(* CODESYS project BelShina_8100_1_1_1.export

Project tree, tasks and I/O mapping:
  application Application
    libraries: ; WagoAppStepper, 1.6.1.1 (WAGO)
    task PLC_Task (cyclic, interval t#50ms, priority 15) calls PLC_PRG
    DataTypes/
      data type ConturBuffer
      data type CurveStates
      data type ForceStepStates
      data type StepperStates
      data type StiffnessTestStates
    GV/
      global variables AI_Sensors
      global variables HMI_Alm
      global variables HMI_Process
      global variables HMI_Stepper
    Program/
      Device/
        Motors/
          ForceStep/
            function block fbForceStep [ST]: METH_Direction
            function block fbGetKoef [ST]
            function block fbSpeedCalc [ST]
            program prForceStep [ST]
          Stepper/
            function block fbStepper [ST]: ACT_MoveHome, ACT_MoveToPos, METH_Direction
            program prLaserStepper_1 [ST]
            program prLaserStepper_2 [ST]
          program prMotion [ST]
        program prDevice [ST]
      IO/
        function block filter [ST]
        function fnoneDigit [ST]
        function fnUpToTen [ST]
        function fnZeroDigit [ST]
        program prInToVars [ST]
      OPC_Sync/
        function block fbReadBuffOPC [ST]
        function block FillBuffer [ST]
      Process/
        GetCurve/
          function block fbGetCurve [ST]
          program prGetCurve_1 [ST]
          program prGetCurve_2 [ST]
          program prGetCurve_2_2 [ST]
        StiffnessTest/
          function block fbCalcDistance [ST]
          function block fbStiffnessTest [ST]
          program prStiffnessTest_1 [ST]
          program prStiffnessTest_2 [ST]
        program prProcess [ST]
      function block LIN_TRAFO [ST]
    Simulation/
      function block fbForceStepSim [ST]
      function block fbStepperSim [ST]
      program prSimulation [ST]
    program PLC_PRG [ST]
    Symbols
*)

// Application/DataTypes/ConturBuffer
TYPE ConturBuffer :
STRUCT
	arStepPos			: ARRAY[0..600] OF REAL;
	arLaserData			: ARRAY[0..600] OF REAL;
	wIndex			: WORD;
	xDone			: BOOL;
	 
END_STRUCT
END_TYPE

// Application/DataTypes/CurveStates

TYPE CurveStates :
(
	CS_Stop 		:= 0,
	CS_Done			:= 1,
	CS_Stopping		:= 2,
	CS_SetStep		:= 3,
	CS_WaitInitial	:= 4,
	CS_SetMeassure	:= 5,
	CS_Measuring	:= 6,
	CS_ReadingOPC	:= 7
);
END_TYPE

// Application/DataTypes/ForceStepStates

TYPE ForceStepStates :
(
	FS_Stop 				:= 0,
	FS_FirstRun 			:= 1,
	FS_WaitRaughApprox		:= 2,
	FS_MakeStep				:= 3,
	FS_CheckForce			:= 4,
	FS_Done					:= 5,
	FS_StartRelease			:= 6,
	FS_WaitRelease			:= 7,
	FS_MovePos				:= 8,
	FS_WaitVelicity			:= 9,
	FS_VelicityMode			:= 10,
	FS_VelicityStopping		:= 11
);
END_TYPE

// Application/DataTypes/StepperStates

TYPE StepperStates :
(
	SM_Idle 			:=0,
	SM_Homing			:=1,
	SM_HommingRough		:=2,
	SM_Home				:=3,
	SM_SetZeroPos		:=4,
	SM_SetPrm			:=5,
	SM_MovingToPos		:=6,
	SM_OnPos			:=7,
	SM_Stopping 		:=8,
	SM_Stop 			:=9
);
END_TYPE

// Application/DataTypes/StiffnessTestStates

TYPE StiffnessTestStates :
(
	ST_Proc_Stop 			:= 0,
	ST_Proc_GettingForce 	:= 1,
	ST_Proc_GettingHalfKoef	:= 2,
	ST_Proc_CalcKoef		:= 3,
	ST_Proc_GettingCurve	:= 4,
	ST_Proc_Done			:= 5,
	ST_Proc_Releasing		:= 6,
	ST_Proc_Stopping		:= 7,
	ST_Proc_GettingFirstCurve:=8,
	ST_Proc_Pause			:= 9,
	ST_SendingData			:=10
	
);
END_TYPE

// Application/GV/AI_Sensors

VAR_GLOBAL
	AI_Rol_1 		AT %IW1 : WORD;
	AI_Rol_2 		AT %IW2 : WORD;
	AI_Laser_1 		AT %IW3 : WORD;
	AI_Laser_2 		AT %IW4 : WORD;
	
	wCounter_1		AT %IW29 : WORD;
	wCounter_2		AT %IW31 : WORD;
	dwCounter		: DWORD;
	Force_Us		AT %IW32 : WORD;
	Force_Ref		AT %IW33 : WORD;
	
	FS_Status_1_1		AT %IB41 : BYTE;
	FS_Status_1_2		AT %IB42 : BYTE;
	FS_Status_1_3		AT %IB43 : BYTE;
	
	FS_Status_Force_3		AT %IB29 : BYTE;
	FS_Status_Force_3_2		AT %IB31 : BYTE;
	
	FS_Status_2_1		AT %IB53 : BYTE;
	FS_Status_2_2		AT %IB54 : BYTE;
	FS_Status_2_3		AT %IB55 : BYTE;
	
	Contr_0		AT %QB38 : BYTE;
	Contr_1		AT %QB42 : BYTE;
	SetPos		AT %QW20 : WORD;
	
	
	
	xStopSwitchLeft: BOOL;
	xStopSwitchRight: BOOL;
	
	LaserHome_1: BOOL;
	LaserHome_2: BOOL;
	LaserUp_1: 	BOOL;
	LaserUp_2:	BOOL;
	
	
	xGlWrite1		:BOOL;
	xGlWrite2		:BOOL;
	
END_VAR

// Application/GV/HMI_Alm

VAR_GLOBAL
	xResetAlm		: BOOL;
	wForceStepAlm	: WORD;
	wAnyAlm			: WORD;
	wAlmLaser_1		: WORD;
	wAlmLaser_2		: WORD;
END_VAR

// Application/GV/HMI_Process

VAR_GLOBAL
	///////////////////////////   GET CURVE 1  //////////////////////
	
	xGC_Start_1: BOOL;
	wGS_State_1: WORD;
	
	///////////////////////////   GET CURVE 2  //////////////////////
	
	xGC_Start_2: BOOL;
	wGS_State_2: WORD;
	
	////////////////////////////  STIFFNESS TEST 1 /////////////////////////////
	
	xGS_StartProc_1: BOOL;
	wST_State_1: WORD;
	rST_Koef_1: REAL;
	wST_HalfPos_1: REAL;
	wST_HalfForce_1: REAL;
	xST_Ready_1: BOOL;
	rST_Way_1:REAL;
	rST_Force_1: REAL;
	xStartAllCurves:	BOOL;
	
	////////////////////////////  STIFFNESS TEST 2 /////////////////////////////
	
	xGS_StartProc_2: BOOL;
	wST_State_2: StiffnessTestStates;
	rST_Koef_2: REAL;
	wST_HalfPos_2: REAL;
	wST_HalfForce_2: REAL;
	xST_Ready_2: BOOL;
	rST_Way_2:REAL;
	rST_Force_2: REAL;
	
	////////////////////////////  STIFFNESS TEST 3 /////////////////////////////
	
	xGS_StartProc_3: BOOL;
	wST_State_3: StiffnessTestStates;
	rST_Koef_3: REAL;
	wST_HalfPos_3: REAL;
	wST_HalfForce_3: REAL;
	xST_Ready_3: BOOL;
	rST_Way_3:REAL;
	rST_Force_3: REAL;
	
	////////////////////////////  DISTANCE /////////////////////////////
	
	rDistance_1		: REAL;
	rDistance_2		: REAL;
	
	rTablePos_1		: REAL;
	rTablePos_2		: REAL;
	rLaserDistance_1		: REAL;
	rLaserDistance_2		: REAL;
	
	xProcFinished			: BOOL;
	wProcType	: WORD;
	xReadOPC_1:	BOOL;
	xReadOPC_2:	BOOL;
	xCurveStarted_1: BOOL;
	xCurveStarted_2: BOOL;
	
	rStepPos_1:	REAL;
	rStepPos_2:	REAL;
	
	rLaserData_1: REAL;
	rLaserData_2: REAL;
	
	wBufferState_1:	WORD;
	wBufferState_2:	WORD;
	
	xContinue:	BOOL;
	
	rRealGetForce:	REAL;
	rRealGetForceMax:	REAL;
	diDistanceForce:	DINT;
	
END_VAR
VAR_GLOBAL RETAIN
	///////////////////////////   GET CURVE 1  //////////////////////
	
	wGC_Distance_1: WORD;
	wGC_InitialPos_1: WORD;
	wGC_EndPos_1: WORD;
	
	///////////////////////////   GET CURVE 2  //////////////////////
	
	wGC_Distance_2: WORD;
	wGC_InitialPos_2: WORD;
	wGC_EndPos_2: WORD;
	
	////////////////////////////  STIFFNESS TEST 1 /////////////////////////////
	
	rST_GetForce_1: REAL;
	rST_SetForce_1: REAL;
	wGS_WaitTillDone_1: WORD;
	
	////////////////////////////  STIFFNESS TEST 2 /////////////////////////////
	
	rST_GetForce_2: REAL;
	rST_SetForce_2: REAL;
	wGS_WaitTillDone_2: WORD;
	
	rKforce_1:	REAL:=1; // попроавка на элластичность троса
	rKforce_2:	REAL:=1; // попроавка на элластичность троса
	rKforce_Ctcle:	REAL:=1; // попроавка на элластичность троса
	rRadius:	REAL:=1;
	
	
	
	wTyreSizeFirst:	WORD;
	wTyreSizeAfter:	WORD;
	
	rCycleForceOffset:	REAL;
	rLineForceOffset_1:	REAL;
	rLineForceOffset_2:	REAL;
	
	rDistanceBetweenLasers:	REAL:=1300;
	
	rLaserSetPos_1:	REAL;
	rLaserSetpos_2:	REAL;
	
END_VAR

// Application/GV/HMI_Stepper

VAR_GLOBAL
	///////////////////////    FORCE STEP    //////////////////////////////
	rFS_GetForce: REAL;	
	xFS_Start: BOOL;
	xFS_Release: BOOL;
	wFS_State: WORD;
	wFS_ActualPos: DWORD;
	xFS_JogLeft: BOOL;
	xFS_JogRight: BOOL;
	rFS_GetForce_check: REAL;	
	rFS_CycledWay:	REAL;
	rFS_LinedWay_1:	REAL;
	rFS_LinedWay_2:	REAL;
	rAngle: REAL;
	
	
	///////////////////////////   LASER  STEP 1  //////////////////////
	xLS_MoveToPos_1: BOOL;
	xLS_MoveHome_1: BOOL;
	xLS_Stop_1: BOOL;
	wLS_GetPos_1: DINT;
	wLS_StepperState_1: WORD;
	xLS_Initilized_1: BOOL;
	rLS_RealPos_1:	REAL;
	
	///////////////////////////   LASER  STEP 2  //////////////////////
	xLS_MoveToPos_2: BOOL;
	xLS_MoveHome_2: BOOL;
	xLS_Stop_2: BOOL;
	wLS_GetPos_2: DINT;
	wLS_StepperState_2: WORD;
	xLS_Initilized_2: BOOL;
	rLS_RealPos_2:	REAL;
	
	
	
END_VAR
VAR_GLOBAL RETAIN
	
///////////////////////    FORCE STEP    //////////////////////////////
	rFS_SetForce: REAL;
	wFS_RoughApprox: WORD;
	wFS_Step: WORD;
	xFS_DirNeg: BOOL;
	rFS_Sensativity: REAL;
	wFS_SetSpeed: WORD;
	wFS_SetAcceleration: WORD;
	wFS_SetDeceleration: WORD;
	wFS_SetBackSpeed: WORD;
	
	
///////////////////////////   LASER  STEP 1  //////////////////////	
	wLS_SetPos_1: WORD;
	wLS_SetSpeed_1: WORD;
	xLS_DirNeg_1: BOOL;
	wLS_Acceleration_1: WORD;
	wLS_Deceleration_1: WORD;
	xLS_StandStill_1:	BOOL;
	
	///////////////////////////   LASER  STEP 2  //////////////////////	
	wLS_SetPos_2: WORD;
	wLS_SetSpeed_2: WORD;
	xLS_DirNeg_2: BOOL;
	wLS_Acceleration_2: WORD;
	wLS_Deceleration_2: WORD;
	xLS_StandStill_2:	BOOL;
	
	
	k_1: REAL:=0.00763;
	k_2: REAL:=0.00763;
	k_3: REAL:=0.0198;
	k_4: REAL:=0.0198;
	
	StepAngle_1:	REAL:=1.8;
	StepAngle_2:	REAL:=1.8;
	ScrewStep_1:	REAL:=24;
	ScrewStep_2:	REAL:=24;
	
	ScrewStepForce:	REAL:=5;
	
	rReductCoef:	REAL:=1;
	rStepAngleForce:	REAL:=1.8;
	
	rForceSensorScale:	REAL:= 20000;
	
	rEncoderImpulseCount: WORD:=5000;
	
	
	
	
	
	
	
	
	
END_VAR

// Application/PLC_PRG
PROGRAM PLC_PRG
VAR
	tnAlmReset:	TON;
	tnStop_1:	TON;
	tnStop_2:	TON;
END_VAR

prInToVars();
prDevice();
prProcess();
tnAlmReset(IN:=xResetAlm, PT:= T#3S);
IF tnAlmReset.Q THEN
	xResetAlm:= FALSE;
END_IF
tnStop_1(IN:=xLS_Stop_1, PT:= T#3S);
IF tnAlmReset.Q THEN
	xLS_Stop_1:= FALSE;
END_IF
tnStop_2(IN:=xLS_Stop_1, PT:= T#3S);
IF tnAlmReset.Q THEN
	xLS_Stop_2:= FALSE;
END_IF
//xResetAlm:=FALSE;
//prSimulation();
//xLS_Stop_1

END_PROGRAM

// Application/Program/IO/prInToVars
PROGRAM prInToVars
	
VAR
	
	_LaserDistance_1: REAL;
	_LaserDistance_2: REAL;
	TRAFO:LIN_TRAFO;
	TRAFO_1:LIN_TRAFO;
	Ud : REAL;
	Uv:	REAL;
	
	filter_1: filter;
	filter_2: filter;
	filter_force: filter;
	k1:	REAL:=0.97;
	k2: REAL:=0.9;
	k_force:REAL:=0.9;
	xSetZero: BOOL;
	rtForceStart:	R_TRIG;
	rtScanStart:	R_TRIG;
	ftContinue:	F_TRIG;
	rtRead1:	F_TRIG;
	rtRead2:	F_TRIG;
	xRef:	BOOL;
	rForceLoc:	REAL;
	rtGetInitialPos:	R_TRIG;
	rOldDistance:	real;
END_VAR

//rDistance_1 := TO_REAL(AI_Rol_1) * k_1;
//rDistance_2 := TO_REAL(AI_Rol_2) * k_2;

rTablePos_1:= TO_REAL(AI_Rol_1) * k_1;
rTablePos_2:= TO_REAL(AI_Rol_2) * k_2;
rTablePos_1:=fnoneDigit(in:= rTablePos_1);
rTablePos_2:=fnoneDigit(in:= rTablePos_2);
//rLaserDistance_1 := 150 + TO_REAL(AI_Laser_1) * k_3;

//rLaserDistance_2 := 150 + rDistanceBetweenLasers - TO_REAL(AI_Laser_2) * k_3;
rtGetInitialPos(CLK:= wGS_State_1 > CS_WaitInitial AND wGS_State_2 > CS_WaitInitial,);
(*IF rtGetInitialPos.Q THEN
	rDistanceBetweenLasers:= (150 + TO_REAL(AI_Laser_1) * k_3) + (150 + TO_REAL(AI_Laser_2) * k_3) + (rRadius * 2);
END_IF*)
_LaserDistance_1:= 150 + TO_REAL(AI_Laser_1) * k_3;
_LaserDistance_2:= rDistanceBetweenLasers - (TO_REAL(AI_Laser_2) * k_3 + 150) - rLaserSetPos_1 - rLaserSetPos_2;
rtScanStart(CLK:= xStartAllCurves); // xContinue
ftContinue(CLK:=xContinue);
rtRead1(CLK:=wLS_StepperState_1 = SM_OnPos);
rtRead2(CLK:=wLS_StepperState_2 = SM_OnPos);
(*
IF wGS_State_1 = CS_WaitInitial OR  rtRead1.Q OR wST_State_1 = ST_Proc_Done OR wST_State_1 = SM_Stop THEN
	//xGlWrite1:=FALSE;
	//filter_1(F_IN:= rDistance_1);
	filter_1(F_IN:= _LaserDistance_1, k:= k1, F_OUT=> rLaserDistance_1);
END_IF
IF wGS_State_2 = CS_WaitInitial OR rtRead2.Q OR wST_State_1 = ST_Proc_Done OR wST_State_1 = SM_Stop THEN
	//xGlWrite2:=FALSE;
	//filter_2(F_IN:= rDistance_2);
	filter_2(F_IN:= _LaserDistance_2, k:= k1,F_OUT=> rLaserDistance_2);
END_IF
*)
filter_1(F_IN:= _LaserDistance_1, k:= k1, F_OUT=> rLaserDistance_1);
filter_2(F_IN:= _LaserDistance_2, k:= k1,F_OUT=> rLaserDistance_2);
rLaserDistance_1:=fnoneDigit(rLaserDistance_1);
rLaserDistance_2:=fnoneDigit(rLaserDistance_2);

//filter_1(F_IN:= rDistance_1, k:= k1, F_OUT=> rLaserDistance_1);
//filter_2(F_IN:= rDistance_2, k:= k1,F_OUT=> rLaserDistance_2);

TRAFO(
	IN:= TO_REAL(Force_Us), 
	IN_MIN:= 0, 
	IN_MAX:= 30000, 
	OUT_MIN:= 0, 
	OUT_MAX:= 15, 
	OUT=> , 
	ERROR=> );
	filter_force(F_IN:= TRAFO.OUT, k:= k_force, F_OUT=> Ud);
	TRAFO_1(
	IN:= TO_REAL(Force_Ref), 
	IN_MIN:= 0, 
	IN_MAX:= 20000, 
	OUT_MIN:= 0, 
	OUT_MAX:= 10, 
	OUT=> Uv, 
	ERROR=> );

	
CASE wProcType OF
	1:
		rFS_GetForce:= (((Ud/2)/(Uv))*rForceSensorScale + rCycleForceOffset) * rKforce_Ctcle * rRadius;
		rFS_GetForce:=fnUpToTen(rFS_GetForce);
		IF (rFS_CycledWay <> rOldDistance) THEN
			rOldDistance:= rFS_CycledWay;
			diDistanceForce:= TO_DINT(rFS_GetForce) * 10000 + TO_DINT(rFS_CycledWay*100);
		END_IF
		
	2:
		rFS_GetForce:= (((Ud/2)/(Uv))*rForceSensorScale + rLineForceOffset_1)* rKforce_1;
		rFS_GetForce:=fnUpToTen(rFS_GetForce);
		IF (rDistance_1 <> rOldDistance) THEN
			rOldDistance:= rDistance_1;
			diDistanceForce:= TO_DINT(rFS_GetForce) * 10000 + TO_DINT(rDistance_1 *100);
		END_IF
		
	3:
		rFS_GetForce:= (((Ud/2)/(Uv))*rForceSensorScale + rLineForceOffset_2) * rKforce_2;
		rFS_GetForce:=fnUpToTen(rFS_GetForce);
		IF (rDistance_2 <> rOldDistance) THEN
			rOldDistance:= rDistance_2;
			diDistanceForce:= TO_DINT(rFS_GetForce) * 10000 + TO_DINT(rDistance_2 *100);
		END_IF
		
END_CASE
//rFS_GetForce:=fnZeroDigit(in:= rFS_GetForce);
//rRealGetForce:= ((Ud/2)/(Uv))*rForceSensorScale * rKforce_1;
//rRealGetForce:=fnZeroDigit(rRealGetForce);
rRealGetForce:= rFS_GetForce / rRadius;
rRealGetForce:= fnUpToTen(rRealGetForce);
rRealGetForceMax:= rST_Force_1 / rRadius;
rRealGetForceMax:= rRealGetForce;

xLS_StandStill_1:=AI_Sensors.FS_Status_1_2.2;
xLS_StandStill_2:=AI_Sensors.FS_Status_2_2.2;

dwCounter:= wCounter_2 * 68835 + wCounter_1;
rAngle:= ((TO_REAL(dwCounter)) / (TO_REAL(rEncoderImpulseCount)) * 90);
rAngle:=fnoneDigit(rAngle);

//xFS_Start
rtForceStart(CLK:=xGS_StartProc_1);

IF rtForceStart.Q THEN
	SetPos:= 5000;
	Contr_0.2:=TRUE;
ELSE
	Contr_0.2:=FALSE;
END_IF

xRef:= FS_Status_Force_3.1;

(*
xStopSwitchLeft:= NOT FS_Status_Force_3.1;
xStopSwitchRight:= NOT FS_Status_Force_3_2.1;

LaserHome_1:= NOT FS_Status_Force_3.1;
LaserHome_2:= NOT FS_Status_Force_3_2.1;

LaserUp_1:= NOT FS_Status_Force_3.4;
LaserUp_2:= NOT FS_Status_Force_3_2.4;
*)

//xSetZero:=FALSE;

END_PROGRAM

// Application/Program/IO/fnoneDigit
FUNCTION fnoneDigit : REAL
VAR_INPUT
	in: REAL;
END_VAR
VAR
	iBuffer:	INT;
	out:	REAL;
END_VAR

iBuffer:= TO_INT(in * 10);
out:=TO_REAL(iBuffer)/10;
fnoneDigit:=out;

END_FUNCTION

// Application/Program/IO/fnUpToTen
FUNCTION fnUpToTen : REAL
VAR_INPUT
	in: REAL;
END_VAR
VAR
	iBuffer:	INT;
	out:	REAL;
END_VAR

iBuffer:= TO_INT(in/10);
out:=iBuffer*10;
fnUpToTen:=out;

END_FUNCTION

// Application/Program/IO/fnZeroDigit
FUNCTION fnZeroDigit : REAL
VAR_INPUT
	in: REAL;
END_VAR
VAR
	iBuffer:	INT;
	out:	REAL;
END_VAR

iBuffer:= TO_INT(in);
out:=iBuffer;
fnZeroDigit:=out;

END_FUNCTION

// Application/Program/LIN_TRAFO
FUNCTION_BLOCK LIN_TRAFO
VAR_INPUT
	IN: REAL;				(* input value*)
	IN_MIN:REAL;			(* minimum input value *)
	IN_MAX:REAL;			(* maximum input value *)
	OUT_MIN:REAL;		(* corresponding minimum output value *)
	OUT_MAX:REAL;		(* corresponding maximum output value *)
END_VAR
VAR_OUTPUT
	OUT: REAL;			(* output value *)
	ERROR: BOOL;		(* error: IN_MIN = IN_MAX or IN out of interval *)
END_VAR

VAR
	Diff: REAL;
END_VAR

Diff := IN_MAX-IN_MIN;
ERROR := (Diff=0) OR (IN<IN_MIN) OR (IN>IN_MAX);

IF NOT ERROR THEN
	OUT := (IN-IN_MIN)/Diff * (OUT_MAX-OUT_MIN) + OUT_MIN;
END_IF

END_FUNCTION_BLOCK

// Application/Program/IO/filter
FUNCTION_BLOCK filter
VAR_INPUT
	F_IN: REAL;
	k:	REAL:=0.9;
END_VAR
VAR_OUTPUT
	F_OUT: REAL;
END_VAR
VAR

END_VAR

F_OUT:=(1-k)*F_IN+k*F_OUT;

END_FUNCTION_BLOCK

// Application/Program/Device/prDevice
PROGRAM prDevice
VAR
END_VAR

prMotion();

END_PROGRAM

// Application/Program/Device/Motors/prMotion
PROGRAM prMotion
VAR
END_VAR

prForceStep();
prLaserStepper_1();
prLaserStepper_2();

END_PROGRAM

// Application/Program/Device/Motors/ForceStep/prForceStep
PROGRAM prForceStep
VAR
	ForceStep:		fbForceStep;
	//GetKoef: fbGetKoef;
	SpeedCalc:		fbSpeedCalc;
	rRatio:			REAL;
END_VAR

SpeedCalc(
	wProcType:= wProcType, 
	rScrewStep:= ScrewStepForce, 
	rReductCoef:= rReductCoef, 
	rStepAngleForce:= rStepAngleForce, 
	rRadius:= rRadius, 
	wStepSpeedRatio=> rRatio);

IF wFS_SetSpeed = 0 THEN
	wFS_SetSpeed:=1;
END_IF
IF wFS_SetAcceleration = 0 THEN
	wFS_SetAcceleration:=1;
END_IF
IF wFS_SetDeceleration = 0 THEN
	wFS_SetDeceleration:= 1;
END_IF

ForceStep(
	rSetForce:= rFS_SetForce, 
	rGetForce:= rFS_GetForce, 
	wRoughApprox:= wFS_RoughApprox, 
	wStep:= wFS_Step, 
	xDirNeg:= true,//xFS_DirNeg, 
	rSensativity:= rFS_Sensativity, 
	wSpeed:= wFS_SetSpeed * TO_WORD(rRatio),
	wFS_SetBackSpeed:= wFS_SetBackSpeed * TO_WORD(rRatio), 
	wAcceleration:= wFS_SetAcceleration * TO_WORD(rRatio), 
	wDeceleration:= wFS_SetDeceleration * TO_WORD(rRatio), 
	I_Port:= IoConfig_Globals.Servo_Stepper_Controller_55_VDC_7_5A, 
	xStart:= xFS_Start,
	xStopSwitchLeft:= xStopSwitchLeft,
	xStopSwitchRight:= xStopSwitchRight,  
	xResetErr:= xResetAlm, 
	xRelease:= xFS_Release,
	xJogLeft:= xFS_JogLeft, 
	xJogRight:= xFS_JogRight,
	wState=> wFS_State,
	wAlm=> wForceStepAlm, 
	diActualPosition=> );
	
	wFS_ActualPos:= ForceStep.diActualPosition;
	
	(*
	GetKoef(
	rCyclePos:= rAngle, 
	rLinePos_1:= rDistance_1, 
	rLinePos_2:= rDistance_2, 
	wForceState:= wFS_State, 
	rGetForce:= rFS_GetForce, 
	wProcType:= wProcType, 
	xStartProc:= xFS_Start, 
	rSetForce:= rFS_SetForce, 
	rK_1:= 0.072, 
	rK_2:= , 
	rK_3:= , 
	KoefCycle=> rST_Koef_1, 
	KoefLine_1=> rST_Koef_2, 
	KoefLine_2=> rST_Koef_3, 
	HalfWayCycle=> wST_HalfPos_1, 
	HalfWayLine_1=> wST_HalfPos_2, 
	HalfWayLine_2=> wST_HalfPos_3, 
	HalfForceCycle=> wST_HalfForce_1, 
	HalfForceLine_1=> wST_HalfForce_2, 
	HalfForceLine_2=> wST_HalfForce_3, 
	WayCycle=> rST_Way_1, 
	WayLine_1=> rST_Way_2, 
	WayLine_2=> rST_Way_3, 
	MaxForce_1=> rST_Force_1,
	MaxForce_2=> rST_Force_2,
	MaxForce_3=> rST_Force_3


);*)

END_PROGRAM

// Application/Program/Device/Motors/ForceStep/fbForceStep
FUNCTION_BLOCK fbForceStep
VAR_INPUT
	rSetForce:			REAL;
	rSetPos:			DINT;
	rGetForce:			REAL;
	wRoughApprox:		WORD;
	wStep:				WORD;
	xDirNeg:			BOOL;
	rSensativity:		REAL;
	wSpeed: 			WORD;
	wFS_SetBackSpeed: 	WORD;
	wAcceleration: 		WORD;
	wDeceleration: 		WORD;
	I_Port: 			WagoAppStepper.WagoTypesModule_75x_67x.I_Module_75x_67x;
	xStopSwitchLeft:		BOOL;
	xStopSwitchRight:		BOOL;
	
END_VAR
VAR_IN_OUT
	xStart:				BOOL;
	xResetErr:			BOOL;
	xRelease:			BOOL;
	xJogLeft:			BOOL;
	xJogRight:			BOOL;
END_VAR
VAR_OUTPUT
	wState:				ForceStepStates;
	diActualPosition: 	DINT;
	wAlm:				WORD;
END_VAR
VAR
	rtStart:			R_TRIG;
	ftStart:			F_TRIG;
	ftRelease:			F_TRIG;
	ControlBasic:		WagoAppStepper.FbStepperControlBasic;
	xEnable: 			BOOL;
	eJobType: 			WagoAppStepper.eMode;
	xTriggerStart: 		BOOL;
	xTriggerErrorReset: BOOL;
	xStop: 				BOOL;
	
	
	diPosition: 		DINT;
	iSpeed: 			INT;
	xJobFinished: 		BOOL;
	xBusy: 				BOOL;
	xError: 			BOOL;
	oStatus: 			WagoAppStepper.WagoSysErrorBase.FbResult;
	eErrorCodes: 		WagoAppStepper.eStatus;
	diRoughDistance:	DINT;
	rCompareForce:		REAL;
	rDirection:			INT;
	rtRelease:			R_TRIG;
	rtJogLeft:			R_TRIG;
	rtJogright:			R_TRIG;
	rtLimit:			R_TRIG;
	rtAlm:				R_TRIG;
END_VAR

VAR RETAIN
	diRetainPos: DINT;
END_VAR

rtStart(CLK:=xStart);
ftStart(CLK:=xStart);
rtRelease(CLK:=xRelease);
ftRelease(CLK:=xRelease);
rtJogLeft(CLK:=xJogLeft AND (NOT xStopSwitchLeft));
rtJogright(CLK:=xJogRight AND (NOT xStopSwitchRight));

IF (ftStart.Q OR ftRelease.Q)AND (NOT (wState = FS_Done)) THEN
	xStop			:= TRUE;
	xTriggerStart	:= FALSE;
	xRelease		:= FALSE;	
	wState:=FS_Stop;
END_IF

IF rtRelease.Q THEN
	xStop			:=TRUE;
	xTriggerStart	:= FALSE;
	xJogLeft		:= FALSE;
	xJogRight		:= FALSE;
	wState			:=FS_StartRelease;
END_IF

IF (rtJogLeft.Q OR rtJogright.Q) AND (NOT(wState = FS_Stop OR wState = FS_Done)) THEN
	xJogLeft		:= FALSE;
	xJogRight		:= FALSE;
END_IF


CASE wState OF
	
		FS_Stop, FS_Done:
		
		
				IF rtStart.Q AND (NOT (xStopSwitchLeft OR xStopSwitchRight)) THEN
					diRoughDistance		:= 0;
					xStop				:=FALSE;
					rCompareForce		:= (rSetForce/100)* wRoughApprox;
					METH_Direction(xDirNeg:= xDirNeg);
					IF rSetPos = 0 THEN
						wState			:= FS_FirstRun;
					ELSE
						xEnable			:= TRUE;
						eJobType		:= MoveRelative;
						diPosition		:= rSetPos;
						iSpeed			:= wSpeed;
						xTriggerStart	:= TRUE;
						wState			:= FS_MovePos;
					END_IF					
				END_IF
				
				IF (xJogLeft AND (NOT xStopSwitchLeft)) OR (xJogRight AND (NOT xStopSwitchRight)) THEN
					xEnable			:= TRUE;
					xStop			:=FALSE;
					eJobType		:= VelocityControl;
					METH_Direction(xDirNeg:= xJogLeft);
					IF xJogLeft THEN
						iSpeed			:= (TO_INT(wSpeed)) * rDirection;
					ELSE
						iSpeed			:= (TO_INT(wFS_SetBackSpeed)) * rDirection;
					END_IF
					xTriggerStart	:= TRUE;
					//wState			:= FS_WaitVelicity;
					wState:=FS_VelicityMode;
				END_IF
					
		
		FS_FirstRun:
		
				xEnable			:= TRUE;
				//eJobType		:= MoveRelative;
				//diPosition		:= 200000 * rDirection;
				//iSpeed			:= wSpeed;
				//xTriggerStart	:=TRUE;
				xStop			:=FALSE;
				eJobType		:= VelocityControl;
				METH_Direction(xDirNeg:= TRUE);
				iSpeed			:= (TO_INT(wSpeed)) * rDirection;
				xTriggerStart	:= TRUE;
				wState			:= FS_WaitRaughApprox;
				
				
		FS_WaitRaughApprox:
		
				IF rGetForce > rCompareForce THEN
					xStop	:=TRUE;
					IF wRoughApprox = 100 THEN						
						xStart	:=FALSE;
						wState	:= FS_Done;
					ELSE
						wState	:= FS_MakeStep;
					END_IF										
				END_IF
				
		
		FS_MakeStep:
				
		
				IF xJobFinished AND ControlBasic.iActualSpeed = 0 THEN
					xStop			:=FALSE;
					IF iSpeed < 0 THEN
						iSpeed:= iSpeed * -1;
					END_IF
					diPosition		:= wStep * rDirection;
					eJobType		:= MoveRelative;
					xTriggerStart	:=TRUE;
					wState			:= FS_CheckForce;
				END_IF
				
				
		FS_CheckForce:
		
				
				IF xJobFinished THEN
					IF (rGetForce < rSetForce + rSensativity) AND (rGetForce > rSetForce - rSensativity) THEN
						xStart	:=FALSE;
						wState	:= FS_Done;
					ELSIF rGetForce < rSetForce - rSensativity THEN
						METH_Direction(xDirNeg:= xDirNeg);
						wState	:= FS_MakeStep;
					ELSIF rGetForce > rSetForce + rSensativity THEN
						METH_Direction(xDirNeg:= NOT xDirNeg);
						wState	:= FS_MakeStep;
					END_IF
				END_IF
				
		FS_StartRelease:
		
				IF xJobFinished THEN
					xStop			:=FALSE;
					METH_Direction(xDirNeg:= NOT xDirNeg);
					xEnable			:= TRUE;
					//eJobType		:= MoveRelative;
					//diPosition		:= 200000 * rDirection;
					//iSpeed			:= wSpeed;
					eJobType		:= VelocityControl;
					iSpeed			:= (TO_INT(wFS_SetBackSpeed)) * rDirection;
					xTriggerStart	:=NOT xStopSwitchRight;
					wState			:= FS_WaitRelease;
				END_IF
				
		FS_WaitRelease:
		
				IF rGetForce < 60 THEN
					xStart:= FALSE;
					xStop			:= TRUE;
					xTriggerStart	:= FALSE;
					xRelease		:= FALSE;	
					wState:=FS_Stop;
				END_IF
				
				
		FS_MovePos:
		
				IF xJobFinished THEN
					wState	:= FS_Done;
				END_IF
				
				
		FS_WaitVelicity:
		
				IF NOT xTriggerStart THEN
					wState	:= FS_VelicityMode;
				END_IF
				
				
		FS_VelicityMode:
		
		
				IF rtJogLeft.Q OR rtJogright.Q THEN
					xJogRight		:=rtJogright.Q;
					xJogLeft		:=rtJogLeft.Q;
					METH_Direction(xDirNeg:= xJogLeft);
					iSpeed			:= (TO_INT(wSpeed)) * rDirection;
					xTriggerStart	:= TRUE;
				END_IF
		
				IF NOT (xJogLeft OR xJogRight) THEN
					iSpeed			:= 0;
					xStop			:= TRUE;
					xTriggerStart	:= TRUE;
					wState			:= FS_VelicityStopping;
				END_IF
				
				
		FS_VelicityStopping:
		
				IF ControlBasic.iActualSpeed = 0 AND (NOT xTriggerStart) THEN
					wState			:= FS_Stop;
				END_IF
				

END_CASE





ControlBasic(
	xEnable:= xEnable, 
	I_Port:= I_Port, 
	eJobType:= eJobType, 
	xDirPos:= NOT xDirNeg, 
	xDirNeg:=  xDirNeg, 
	iSpeed:= iSpeed, 
	wAcceleration:= wAcceleration, 
	wDeceleration:= wDeceleration, 
	diPosition:= diPosition, 
	xTriggerStart:= xTriggerStart, 
	xTriggerErrorReset:= xTriggerErrorReset, 
	xStop:= xStop, 
	xJobFinished=> xJobFinished, 
	xBusy=> xBusy, 
	xError=> xError, 
	oStatus=> oStatus, 
	eErrorCodes=> eErrorCodes, 
	diActualPosition=> diActualPosition, 
	iActualSpeed=> , 
	xMailboxActive=> , 
	xResetWarning=> );
	
	IF xError THEN
		wAlm.0:=TRUE;
	ELSE
		xTriggerErrorReset:= FALSE;
		wAlm.0:=FALSE;
	END_IF
	
	IF xResetErr THEN
		xTriggerErrorReset:=TRUE;
		xStop:= FALSE;
		wAlm:=0;
	END_IF

	rtLimit(CLK:=xStopSwitchLeft OR xStopSwitchRight);
	IF rtLimit.Q THEN
		wAlm.1:=TRUE;
	END_IF
	
	rtAlm(CLK:= wAlm > 0);
	IF rtAlm.Q THEN
		xStop:=TRUE;
		wState:= FS_VelicityStopping;
	END_IF

METHOD METH_Direction
VAR_INPUT
	xDirNeg:	BOOL;
END_VAR
IF xDirNeg THEN
	rDirection:= -1;
ELSE
	rDirection:= 1;
END_IF
END_METHOD

END_FUNCTION_BLOCK

// Application/Program/Device/Motors/ForceStep/fbGetKoef
FUNCTION_BLOCK fbGetKoef
VAR_INPUT
	rCyclePos		:	REAL;
	rLinePos_1		:	REAL;
	rLinePos_2		:	REAL;
	wForceState		:	ForceStepStates;
	rGetForce		:	REAL;
	wProcType		:	WORD;
	xStartProc		:	BOOL;
	rSetForce		:	REAL;
	//rGetForce		:	REAL;
	rK_1			:	REAL;
	rK_2			:	REAL;
	rK_3			:	REAL;
END_VAR
VAR_OUTPUT
	KoefCycle:	REAL;
	KoefLine_1:	REAL;
	KoefLine_2:	REAL;
	HalfWayCycle:	REAL;
	HalfWayLine_1:	REAL;
	HalfWayLine_2:	REAL;
	HalfForceCycle:	REAL;
	HalfForceLine_1:	REAL;
	HalfForceLine_2:	REAL;
	WayCycle:		REAL;
	WayLine_1:		REAL;
	WayLine_2:		REAL;
	MaxForce_1:	REAL;
	MaxForce_2:	REAL;
	MaxForce_3:	REAL;
END_VAR
VAR
	rtFirstRun	: R_TRIG;
	ftFirstRun	: F_TRIG;
	rtHalfForce	: R_TRIG;
	rStartPos	: REAL;
END_VAR

rtFirstRun(CLK:=xStartProc);
ftFirstRun(CLK:=xStartProc);
rtHalfForce(CLK:= (xStartProc AND (rGetForce > (rSetForce / 2))));

CASE wProcType OF 
	1:
		IF rtFirstRun.Q THEN
			rStartPos:= rCyclePos;
		END_IF
		
		IF rtHalfForce.Q THEN
			HalfForceCycle:= rGetForce;
			IF rCyclePos > rStartPos THEN
				HalfWayCycle:= (rCyclePos - rStartPos);
			ELSE 
				HalfWayCycle:= (360 - rStartPos + rCyclePos);
			END_IF
		END_IF
		
		IF ftFirstRun.Q THEN
			MaxForce_1:= rGetForce ;
			IF rCyclePos > rStartPos THEN
				WayCycle:= (rCyclePos - rStartPos);
			ELSE 
				WayCycle:= (360 - rStartPos + rCyclePos);
			END_IF
			//KoefCycle:= 
		END_IF
		
	2:
	
		IF rtFirstRun.Q THEN
			rStartPos:= rLinePos_1;
		END_IF
		
		IF rtHalfForce.Q THEN
			HalfForceLine_1:= rGetForce;			
			HalfWayLine_1:= (rStartPos - rLinePos_1);			
		END_IF
		
		IF ftFirstRun.Q THEN
			MaxForce_2:= rGetForce ;
			//HalfForceLine_1:= rGetForce;			
			WayLine_2:= (rStartPos - rLinePos_1);
		END_IF
		
	3:
	
	
		IF rtFirstRun.Q THEN
			rStartPos:= rLinePos_2;
		END_IF
		
		IF rtHalfForce.Q THEN
			HalfForceLine_2:= rGetForce;			
			HalfWayLine_2:= (rStartPos - rLinePos_2);			
		END_IF
		
		IF ftFirstRun.Q THEN
			MaxForce_3:= rGetForce ;
			//HalfForceLine_2:= rGetForce;			
			WayLine_2:= (rStartPos - rLinePos_2);
		END_IF
			
END_CASE

END_FUNCTION_BLOCK

// Application/Program/Device/Motors/ForceStep/fbSpeedCalc
FUNCTION_BLOCK fbSpeedCalc
VAR_INPUT
	
	wProcType			: WORD;
	rScrewStep			: REAL:=5;
	rReductCoef			: REAL:=1;
	rStepAngleForce		: REAL:=1.8;
	rRadius				: REAL:=1;
END_VAR
VAR_OUTPUT
	wStepSpeedRatio			: REAL;			
END_VAR
VAR
	rMotorSteps			: REAL;
	rCycleMM			: REAL;
	rLineSpeedRatio			: REAL;
END_VAR

rMotorSteps	:= 23040/rStepAngleForce;
rCycleMM	:= rReductCoef/rScrewStep;
rLineSpeedRatio	:= rMotorSteps * rCycleMM;
(*IF wProcType = 1 THEN
	wStepSpeedRatio	:= rLineSpeedRatio;
ELSE
	wStepSpeedRatio	:= (360 * rLineSpeedRatio)/(200 * 3.14 * rRadius);
END_IF
*)
wStepSpeedRatio	:= rLineSpeedRatio/60;

END_FUNCTION_BLOCK

// Application/Program/Device/Motors/Stepper/prLaserStepper_1
PROGRAM prLaserStepper_1
VAR
	LaserStepper	:	fbStepper;
	xMoveRelative	: 	BOOL;
	wRatio			: 	word;
	xCheck: bool;
		
	xTriggerErrorReset: BOOL;
END_VAR

wRatio:= TO_WORD(((360 / StepAngle_1) * 64) / ScrewStep_1);

IF wLS_SetSpeed_1 = 0 THEN
	wLS_SetSpeed_1:=1;
END_IF
IF wLS_Acceleration_1 = 0 THEN
	wLS_Acceleration_1:=1;
END_IF
IF wLS_Deceleration_1 = 0 THEN
	wLS_Deceleration_1:=1;
END_IF

IF xResetAlm THEN
	xTriggerErrorReset:=TRUE;
END_IF

LaserStepper(
	diSetPos:= wLS_SetPos_1 * wRatio, 
	xMoveRelative:= xMoveRelative, 
	wSetSpeed:= (wLS_SetSpeed_1 * wRatio) / 60,
	xHomeIn:= LaserHome_1,//(AI_Laser_1 > 1200) AND (AI_Laser_1 < 1600),
	xLaserUp:= LaserUp_1, 
	xDirNeg:= xLS_DirNeg_1, 
	wAcceleration:= (wLS_Acceleration_1 * wRatio) / 60, 
	wDeceleration:= (wLS_Deceleration_1 * wRatio) / 60, 
	I_Port:= IoConfig_Globals.Servo_Stepper_Controller_55_VDC_7_5A_1, 
	xMoveToPos:= xLS_MoveToPos_1,
	xTriggerErrorReset:=xTriggerErrorReset, 
	xMoveHome:= xLS_MoveHome_1, 
	xStop:= xLS_Stop_1, 
	diGetPos=> ,
	wAlmLaser=> wAlmLaser_1, 
	xInitilized=> xLS_Initilized_1, 
	wStepperState=> wLS_StepperState_1);
	
	//wAlmLaser_1
	
	wLS_GetPos_1:=LaserStepper.diGetPos/wRatio;
	rLS_RealPos_1:=TO_REAL(LaserStepper.diGetPos)/wRatio;
	IF xLS_StandStill_1 THEN
		xCheck:= true;
	END_IF

END_PROGRAM

// Application/Program/Device/Motors/Stepper/fbStepper
FUNCTION_BLOCK fbStepper
VAR_INPUT
	diSetPos:			DINT;
	xMoveRelative:		BOOL;
	wSetSpeed:			WORD;
	xDirNeg:			BOOL;
	wAcceleration: 		WORD;
	wDeceleration: 		WORD;
	I_Port: 			WagoAppStepper.WagoTypesModule_75x_67x.I_Module_75x_67x;
	xHomeIn:	BOOL;
	xLaserUp:	BOOL;
	
END_VAR
VAR_IN_OUT
	xMoveToPos:			BOOL;
	xMoveHome:			BOOL;
	xStop:				BOOL;
	xTriggerErrorReset: BOOL;
END_VAR
VAR_OUTPUT
	diGetPos:			DINT;
	xInitilized:		BOOL;
	wStepperState:		StepperStates;
	wAlmLaser:		WORD;
END_VAR
VAR
	rtMoveToPos:		R_TRIG;
	rtMoveHome:			R_TRIG;
	rtStop:				R_TRIG;
	ControlBasic:		WagoAppStepper.FbStepperControlBasic;
	xEnable: 			BOOL;
	eJobType: 			WagoAppStepper.eMode;
	xTriggerStart: 		BOOL;
	
	iSpeed: 			INT;
	
	diPosition: 		DINT;
	
	xJobFinished: 		BOOL;
	xBusy: 				BOOL;
	xError: 			BOOL;
	oStatus: 			WagoAppStepper.WagoSysErrorBase.FbResult;
	eErrorCodes: 		WagoAppStepper.eStatus;
	diRoughDistance:	DINT;
	rCompareForce:		REAL;
	rDirection:			INT;
	iActualSpeed: INT;
	SetPosition:WagoAppStepper.FbSetPosition;
	xSetZeroPos: BOOL;
	xHome: BOOL;
	rtHome:	R_TRIG;
	xStopLoc: BOOL;
	iSetSpeed: INT;
	xDirNegLoc: BOOL;
	tnWait			:	TON;
	rtUp			:	R_TRIG;
	ftHome			:	F_TRIG;
	rtSet			:	R_TRIG;
	tnWaitSetPos	:	TON;
END_VAR

rtMoveToPos(CLK:=xMoveToPos);
rtMoveHome(CLK:=xMoveHome AND (NOT xLaserUp));
rtStop(CLK:=xStop);

IF rtMoveHome.Q AND NOT xInitilized THEN	
	wStepperState:= SM_Idle;
END_IF

IF rtStop.Q THEN
	xStopLoc		:= TRUE;
	
	xMoveToPos		:= FALSE;
	xMoveHome		:= FALSE;
	wStepperState	:= SM_Stopping;
END_IF


CASE wStepperState OF
	
		
			SM_Idle:
			
								
				IF rtMoveToPos.Q OR rtMoveHome.Q THEN
					ACT_MoveHome();					
				END_IF
				
				IF xBusy AND iActualSpeed <> 0 AND (xMoveToPos OR xMoveHome) THEN
					wStepperState	:= SM_HommingRough;
				END_IF
				
				
			SM_HommingRough:
			
				IF xHomeIn THEN
					//METH_Direction(xDirNeg:= xDirNeg);
					xEnable			:= TRUE;
					xDirNegLoc		:= NOT xDirNeg;
					//xStopLoc		:= FALSE;
					iSetSpeed		:=200;
					eJobType		:= VelocityControl;
					xTriggerStart	:=TRUE;
					wStepperState	:= SM_Homing;
				END_IF
				
				
			SM_Homing:
			
				(*IF xBusy AND iActualSpeed = 0 THEN
					xStopLoc:= TRUE;
				END_IF
				IF NOT xBusy THEN
					xStopLoc	:= FALSE;
					xSetZeroPos	:= TRUE;
				END_IF*)
				ftHome(CLK:=xHomeIn);
				IF ftHome.Q THEN
					//xSetZeroPos		:= FALSE;
					xStopLoc		:= TRUE;
					//xInitilized		:= TRUE;
					xMoveHome		:= FALSE;
					tnWait(IN:=FALSE);
					wStepperState	:= SM_SetZeroPos;
				END_IF
				
			
			SM_SetZeroPos:
			
				IF NOT xBusy THEN
					xStopLoc	:= FALSE;
				END_IF
				
				tnWait(IN:=NOT xStopLoc, PT:=T#2S);
				IF tnWait.Q THEN
					tnWait(IN:=FALSE);
					xSetZeroPos	:= TRUE;
					wStepperState	:= SM_Home;					
				END_IF
				 
			
			SM_Stop: 					
				
				IF xMoveToPos AND ((NOT xLaserUp) OR (diGetPos > diSetPos)) THEN
					ACT_MoveToPos();					
				END_IF
				
			SM_Home:
			
				tnWaitSetPos(IN:= xHome, PT:= T#2S);
				IF tnWaitSetPos.Q THEN
					tnWaitSetPos(IN:= FALSE);
					xSetZeroPos	:= FALSE;
					xInitilized	:= TRUE;
				END_IF
				
				tnWait(IN:=NOT xSetZeroPos, PT:=T#2S);
				IF xMoveToPos AND tnWait.Q THEN
					tnWait(IN:=FALSE);
					ACT_MoveToPos();					
				END_IF
				
			
				
			SM_OnPos: 
			
				IF xMoveToPos AND ((NOT xLaserUp) OR (diGetPos > diSetPos))  THEN
					//tnWait(IN:=FALSE);
					ACT_MoveToPos();					
				END_IF
				
				
			SM_SetPrm:
			
				IF xBusy THEN
					//xTriggerStart	:=FALSE;
					wStepperState	:= SM_MovingToPos;
				END_IF
				
				
			SM_MovingToPos:
			
				tnWait(IN:=xJobFinished, PT:=T#1S);
				IF (*tnWait.Q*)  xJobFinished  THEN
					tnWait(IN:=FALSE);
					xMoveToPos		:=FALSE;
					wStepperState	:= SM_OnPos;
				END_IF
				
				
			SM_Stopping:
			
				IF iActualSpeed = 0 THEN
					//xStopLoc		:= FALSE;
					//xStop			:= FALSE;
					IF xInitilized THEN
						wStepperState	:= SM_Stop;
					ELSE
						wStepperState	:= SM_Idle;
					END_IF
				END_IF
				
END_CASE

rtUp(CLK:=xLaserUp);

IF rtUp.Q THEN
	xStopLoc:= TRUE;
	wAlmLaser.1:= TRUE;
	wStepperState:= SM_Stopping;
END_IF

IF xTriggerErrorReset THEN
	xSetZeroPos:=FALSE;
	wAlmLaser:= 0;
	//xStopLoc:= xEnable;
END_IF
ControlBasic(
	xEnable:= xEnable, 
	I_Port:= I_Port, 
	eJobType:= eJobType, 
	xDirPos:= NOT xDirNeg, 
	xDirNeg:= xDirNegLoc,//xDirNeg, 
	iSpeed:= iSetSpeed, 
	wAcceleration:= wAcceleration, 
	wDeceleration:= wDeceleration, 
	diPosition:= diPosition, 
	xTriggerStart:= xTriggerStart, 
	xTriggerErrorReset:= xTriggerErrorReset, 
	xStop:= xStopLoc, 
	xJobFinished=> xJobFinished, 
	xBusy=> xBusy, 
	xError=> xError, 
	oStatus=> oStatus, 
	eErrorCodes=> eErrorCodes, 
	diActualPosition=> diGetPos, 
	iActualSpeed=> iActualSpeed, 
	xMailboxActive=> , 
	xResetWarning=> );
	
	IF xError THEN
		wAlmLaser.0:= TRUE;
	ELSE
		wAlmLaser.0:= FALSE;
		xTriggerErrorReset:= FALSE;
	END_IF
	

SetPosition(
	xExecute:= xSetZeroPos, 
	I_Port:= I_Port, 
	diPosition:= 60, 
	xDone=> xHome, 
	xBusy=> , 
	xError=> , 
	oStatus=> );

ACTION ACT_MoveHome:
	//METH_Direction(xDirNeg:= NOT xDirNeg);
	xEnable			:= TRUE;
	xStopLoc		:= FALSE;
	eJobType		:= VelocityControl;//MoveRelative;
	iSetSpeed		:=  wSetSpeed;
	xDirNegLoc		:= NOT xDirNeg;
	//diPosition		:= 200000 * rDirection;
	xTriggerStart	:=TRUE;
END_ACTION

ACTION ACT_MoveToPos:
	METH_Direction(xDirNeg:= xDirNeg);
	xStopLoc			:= FALSE;
	xEnable			:= TRUE;					
	eJobType		:= MoveAbsolute;
	diPosition		:= diSetPos;
	iSetSpeed		:= wSetSpeed;
	xDirNegLoc		:= xDirNeg;
	xTriggerStart	:=TRUE;
	wStepperState	:= SM_SetPrm;
END_ACTION

METHOD METH_Direction
VAR_INPUT
	xDirNeg:	BOOL;
END_VAR
IF xDirNeg THEN
	rDirection:= -1;
ELSE
	rDirection:= 1;
END_IF
END_METHOD

END_FUNCTION_BLOCK

// Application/Program/Device/Motors/Stepper/prLaserStepper_2
PROGRAM prLaserStepper_2
VAR
	LaserStepper	:	fbStepper;
	xMoveRelative	: 	BOOL;
	wRatio			: 	WORD;
	xTriggerErrorReset: BOOL;
END_VAR

wRatio:= TO_WORD(((360 / StepAngle_2) * 64) / ScrewStep_2);

IF wLS_SetSpeed_2 = 0 THEN
	wLS_SetSpeed_2:=1;
END_IF
IF wLS_Acceleration_2 = 0 THEN
	wLS_Acceleration_2:=1;
END_IF
IF wLS_Deceleration_2 = 0 THEN
	wLS_Deceleration_2:=1;
END_IF

IF xResetAlm THEN
	xTriggerErrorReset:=TRUE;
END_IF

LaserStepper(
	diSetPos:= wLS_SetPos_2 * wRatio, 
	xMoveRelative:= xMoveRelative, 
	wSetSpeed:= (wLS_SetSpeed_2 * wRatio)/60,
	xHomeIn:= LaserHome_2,//(AI_Laser_2 > 2000) AND (AI_Laser_2 < 2600),
	xLaserUp:= LaserUp_2,
	xDirNeg:= xLS_DirNeg_2, 
	wAcceleration:= (wLS_Acceleration_2 * wRatio)/60 , 
	wDeceleration:= (wLS_Deceleration_2 * wRatio)/60, 
	I_Port:= IoConfig_Globals.Servo_Stepper_Controller_55_VDC_7_5A_2, 
	xMoveToPos:= xLS_MoveToPos_2,
	xTriggerErrorReset:=xTriggerErrorReset, 
	xMoveHome:= xLS_MoveHome_2, 
	xStop:= xLS_Stop_2, 
	diGetPos=> , 
	wAlmLaser=> wAlmLaser_2,
	xInitilized=> xLS_Initilized_2, 
	wStepperState=> wLS_StepperState_2);
	
	wLS_GetPos_2:=LaserStepper.diGetPos/wRatio;
	rLS_RealPos_2:=TO_REAL(LaserStepper.diGetPos)/wRatio;

END_PROGRAM

// Application/Program/Process/prProcess
PROGRAM prProcess
VAR
	rtStartCurves:	R_TRIG;
	ftStartCurves:	F_TRIG;
	rtStopCurves:	R_TRIG;
END_VAR

prGetCurve_1();
prGetCurve_2_2();
prStiffnessTest_1();

rtStartCurves(CLK:=xStartAllCurves);
ftStartCurves(CLK:=xStartAllCurves);
rtStopCurves(CLK:= NOT (xGC_Start_1 OR xGC_Start_2));


IF rtStartCurves.Q THEN
	xGC_Start_1:= TRUE;
	xGC_Start_2:= TRUE;
END_IF
IF ftStartCurves.Q THEN
	xGC_Start_1:= FALSE;
	xGC_Start_2:= FALSE;
END_IF
IF rtStopCurves.Q THEN
	xStartAllCurves:= FALSE;
END_IF

(*prStiffnessTest_2();*)
IF xProcFinished THEN
	xProcFinished:= FALSE;
END_IF

IF xResetAlm THEN
	//xResetAlm		:= false;
	wForceStepAlm	:= 0;
	wAnyAlm			:= 0;
	wAlmLaser_1		:= 0;
	wAlmLaser_2		:= 0;
END_IF

END_PROGRAM

// Application/Program/Process/GetCurve/prGetCurve_1
PROGRAM prGetCurve_1
VAR
	GetCurve	: fbGetCurve;
	FillBuffer_	: FillBuffer;	
	xStartFilling: BOOL;
	xStopFilling: BOOL;
	xWrite: BOOL;
	xStartSending: BOOL;
	ConturBuffer_:	ConturBuffer;
	rtStopFilling:	R_TRIG;
	rtStartFilling:	R_TRIG;
	rtStopSending:	R_TRIG;
	ReadBuffOPC: fbReadBuffOPC;
	xStopSending: BOOL;
	ftStartProc:	F_TRIG;
END_VAR


GetCurve(
	diDistance:= wGC_Distance_1,
	rGetPos:= rLS_RealPos_1, 
	wStepperState:= wLS_StepperState_1, 
	xInitilized:= xLS_Initilized_1, 
	wInitialPos:= wGC_InitialPos_1,
	wCoupledState:= wGS_State_2,
	xReadOPC:=	xWrite,//wGC_InitialPos_1, xReadOPC_1 
	wEndPos:= wGC_EndPos_1,
	xCurveStarted:=xCurveStarted_1, 
	xStart:= xGC_Start_1, 
	xMovePos:= xLS_MoveToPos_1, 
	xStopStep:= xLS_Stop_1, 
	wSetPos:= wLS_SetPos_1, 
	wState=> wGS_State_1);
	IF xWrite THEN
		xGlWrite1:=TRUE;
	END_IF

rtStopFilling(CLK:=xCurveStarted_1);	
IF rtStopFilling.Q THEN
	xStartFilling:=	TRUE;
END_IF

rtStopFilling(CLK:=wGS_State_1 = CS_Done);
IF rtStopFilling.Q THEN
	xStopFilling:= TRUE;
END_IF

rtStopSending(CLK:=(wGS_State_1 = CS_Stop) OR (NOT xGS_StartProc_1));
IF rtStopSending.Q THEN
	xStopSending:=TRUE;
END_IF
	
FillBuffer_(
	rStepPos:= rLS_RealPos_1 - wGC_InitialPos_1, 
	rLaserData:= rLaserDistance_1, 
	xStart:= xStartFilling, 
	xStop:= xStopFilling, 
	xWrite:= xWrite,
	xStartSending:= xStartSending,  
	ConturBuffer=> ConturBuffer_);
	

ReadBuffOPC(
	ConturBuffer:= ConturBuffer_, 
	wIndexOfReadynnes:= 5, 
	xStart:= xStartSending, 
	xSend:= xReadOPC_1,
	xStop:= xStopSending, 
	rStepPos=> rStepPos_1, 
	rLaserData=> rLaserData_1, 
	wState=> wBufferState_1);

END_PROGRAM

// Application/Program/Process/GetCurve/fbGetCurve
FUNCTION_BLOCK fbGetCurve
VAR_INPUT
	rGetPos			: REAL;
	diDistance		: DINT;
	wStepperState	: StepperStates;
	xInitilized		: BOOL;
	wInitialPos		: WORD;
	wEndPos			: WORD;
	wStepsNomber	: WORD:=100;
	wCoupledState	: CurveStates;
END_VAR
VAR_IN_OUT
	xStart			: BOOL;
	xMovePos		: BOOL;
	xStopStep		: BOOL;
	wSetPos			: WORD;
	xReadOPC		: BOOL;
	xCurveStarted	: bool;
END_VAR
VAR_OUTPUT
	wState			: CurveStates;	
END_VAR
VAR
	rtStart			: R_TRIG;
	ftStart			: F_TRIG;
	tnWait			:	TON;
	wStep			: WORD;
END_VAR

rtStart(CLK:= xStart);
ftStart(CLK:= xStart);

IF ftStart.Q AND (NOT (wState = CS_Done))THEN
	xStopStep:= TRUE;
	wState:= CS_Stop;
END_IF

wStep:= wEndPos/wStepsNomber;
IF wStep = 0 THEN
	wStep := 1;
END_IF

CASE wState OF
	

		CS_Stop, CS_Done:
		
			IF xStart THEN
				xMovePos		:= TRUE;
				wSetPos			:= wInitialPos;
				xCurveStarted	:= TRUE;
				wState			:= CS_SetStep;
			END_IF
			
			
		CS_SetStep:
		
			IF wStepperState = SM_MovingToPos THEN
				tnWait(IN:=FALSE);
				wState		:= CS_WaitInitial;
			END_IF
			
		CS_WaitInitial:
		
			tnWait(IN:=wStepperState = SM_OnPos AND (wCoupledState >= CS_WaitInitial) AND (NOT xCurveStarted), pt:=T#20S);
			IF tnWait.Q THEN
				tnWait(IN:=FALSE);
				//xMovePos	:= TRUE;
				//wSetPos		:= wInitialPos + wStep;
				//wState		:= CS_SetMeassure;
				xReadOPC		:= TRUE;
				wState			:= CS_ReadingOPC;
			END_IF
			
		CS_SetMeassure:
		
			IF wStepperState = SM_MovingToPos  THEN
				wState		:= CS_Measuring;
			END_IF 
				
		CS_Measuring:
			
			tnWait(IN:= wStepperState = SM_OnPos, PT:=T#2S);	
			IF tnWait.Q THEN
				tnWait(IN:= FALSE);
				xReadOPC	:= TRUE;
				wState		:= CS_ReadingOPC;
			END_IF
			
			
		CS_ReadingOPC:
		
			//tnWait(IN:= NOT xReadOPC, PT:=T#3S);
			IF (*tnWait.Q*) NOT xReadOPC THEN
				//tnWait(IN:= FALSE);
				IF rGetPos > wEndPos + wInitialPos THEN
					xStart		:= FALSE;
					xMovePos	:= TRUE;
					wSetPos		:= wInitialPos;
					wState		:= CS_Done;
				ELSE
					xMovePos	:= TRUE;
					wSetPos		:= TO_WORD(rGetPos + wStep);
					wState		:= CS_SetMeassure;
				END_IF
			END_IF
			
	


END_CASE

END_FUNCTION_BLOCK

// Application/Program/OPC_Sync/FillBuffer
FUNCTION_BLOCK FillBuffer
VAR_INPUT
	rStepPos			: REAL;
	rLaserData			: REAL;
	
END_VAR
VAR_IN_OUT
	xStart				: BOOL;
	xStop				: BOOL;
	xWrite				: BOOL;
	xStartSending		: bool;
END_VAR
VAR_OUTPUT
	ConturBuffer		: ConturBuffer;
END_VAR
VAR
END_VAR

IF xStart THEN
	xStart				:= FALSE;
	xStartSending		:= TRUE;
	ConturBuffer.wIndex	:= 0;
	ConturBuffer.xDone	:= FALSE;
	
END_IF

IF xStop THEN
	xStop				:= FALSE;
	ConturBuffer.xDone	:= TRUE;
END_IF

IF xWrite AND (rStepPos = 0 OR rStepPos > 0)THEN
	xWrite:=FALSE;
	ConturBuffer.arLaserData[ConturBuffer.wIndex] 	:= rLaserData;
	ConturBuffer.arStepPos[ConturBuffer.wIndex] 	:= rStepPos;
	ConturBuffer.wIndex								:= ConturBuffer.wIndex + 1;				
END_IF

END_FUNCTION_BLOCK

// Application/Program/OPC_Sync/fbReadBuffOPC
FUNCTION_BLOCK fbReadBuffOPC
VAR_INPUT
	ConturBuffer		: ConturBuffer;
	wIndexOfReadynnes	: WORD:= 5;
END_VAR
VAR_IN_OUT
	xStart				: BOOL;
	xStop				: BOOL;
	xSend				: BOOL;
END_VAR
VAR_OUTPUT
	rStepPos		: REAL;
	rLaserData		: REAL;
	wState			: WORD;
END_VAR
VAR
	tnWait			: TON;
	wIndex			: WORD;
END_VAR

IF xStop THEN
	xStop	:=FALSE;
	xSend	:= 0;
	wState	:= 0;
END_IF

CASE wState OF
	
	0:
		IF xStart THEN
			xStart:= FALSE;
			wIndex:= 0;
			tnWait(IN:= FALSE);
			wState:=1;
		END_IF
		
	1:
		//xStart:= FALSE;
		IF ConturBuffer.wIndex < wIndexOfReadynnes AND (NOT ConturBuffer.xDone) THEN
			wState:=2;
		END_IF
		
	2:
		//xStart:= FALSE;
		IF xStart THEN
			wState:=0;
		END_IF
		IF ConturBuffer.wIndex > wIndexOfReadynnes THEN
			rStepPos		:= ConturBuffer.arStepPos[0];
			rLaserData		:= ConturBuffer.arLaserData[0];
			wState			:=3;
		END_IF
		
	3:
		IF xStart THEN
			wState:=0;
		END_IF
		tnWait(IN:= TRUE, PT:=T#1500MS);
		IF tnWait.Q THEN
			tnWait(IN:= FALSE);
			xSend:=TRUE;
			wState:=4;
		END_IF
		
	4:
		IF xStart THEN
			wState:=0;
		END_IF
		IF (NOT xSend) AND (wIndex < ConturBuffer.wIndex) THEN
			
			rStepPos		:= ConturBuffer.arStepPos[wIndex];
			rLaserData		:= ConturBuffer.arLaserData[wIndex];
			wIndex			:= wIndex + 1;
			wState			:=3;
		ELSIF (NOT xSend) AND (wIndex = ConturBuffer.wIndex) AND ConturBuffer.xDone THEN
			wState			:=0;		 
		END_IF
		
				
END_CASE

END_FUNCTION_BLOCK

// Application/Program/Process/GetCurve/prGetCurve_2_2
PROGRAM prGetCurve_2_2
VAR
	GetCurve	: fbGetCurve;
	FillBuffer_	: FillBuffer;	
	xStartFilling: BOOL;
	xStopFilling: BOOL;
	xWrite: BOOL;
	xStartSending: BOOL;
	ConturBuffer_:	ConturBuffer;
	rtStopFilling:	R_TRIG;
	rtStartFilling:	R_TRIG;
	rtStopSending:	R_TRIG;
	ReadBuffOPC: fbReadBuffOPC;
	xStopSending: BOOL;
END_VAR



GetCurve(
	diDistance:= wGC_Distance_2,
	rGetPos:= rLS_RealPos_2, 
	wStepperState:= wLS_StepperState_2, 
	xInitilized:= xLS_Initilized_2, 
	wInitialPos:= wGC_InitialPos_2,
	wCoupledState:= wGS_State_1,
	xReadOPC:=	xWrite,//wGC_InitialPos_1, xReadOPC_1 
	wEndPos:= wGC_EndPos_1,
	xCurveStarted:=xCurveStarted_2, 
	xStart:= xGC_Start_2, 
	xMovePos:= xLS_MoveToPos_2, 
	xStopStep:= xLS_Stop_2, 
	wSetPos:= wLS_SetPos_2, 
	wState=> wGS_State_2);
	
	IF xWrite THEN
		xGlWrite2:=TRUE;
	END_IF

rtStopFilling(CLK:=xCurveStarted_2);	
IF rtStopFilling.Q THEN
	xStartFilling:=	TRUE;
END_IF

rtStopFilling(CLK:=wGS_State_2 = CS_Done);
IF rtStopFilling.Q THEN
	xStopFilling:= TRUE;
END_IF

rtStopSending(CLK:=(wGS_State_2 = CS_Stop)  OR (NOT xGS_StartProc_1));
IF rtStopSending.Q THEN
	xStopSending:=TRUE;
END_IF
	
FillBuffer_(
	rStepPos:= rLS_RealPos_2 - wGC_InitialPos_2, 
	rLaserData:= rLaserDistance_2, 
	xStart:= xStartFilling, 
	xStop:= xStopFilling, 
	xWrite:= xWrite,
	xStartSending:= xStartSending,  
	ConturBuffer=> ConturBuffer_);

	
ReadBuffOPC(
	ConturBuffer:= ConturBuffer_, 
	wIndexOfReadynnes:= 5, 
	xStart:= xStartSending, 
	xSend:= xReadOPC_2,
	xStop:= xStopSending, 
	rStepPos=> rStepPos_2, 
	rLaserData=> rLaserData_2, 
	wState=> wBufferState_2);

END_PROGRAM

// Application/Program/Process/StiffnessTest/prStiffnessTest_1
PROGRAM prStiffnessTest_1
VAR
	StiffnessTest: fbStiffnessTest;	
	CalcDistance: fbCalcDistance;
END_VAR

StiffnessTest(
	xReady:= xST_Ready_1,
	wTyreSizeFirst:= wTyreSizeFirst, 
	wTyreSizeAfter:= wTyreSizeAfter,
	wBufferState_1:= wBufferState_1,
	wBufferState_2:= wBufferState_2,
	wProcType:= wProcType,
	rGetForce:= rFS_GetForce, 
	rSetForce:= rST_SetForce_1, 
	wGetPos:= wFS_ActualPos,
	rFS_CycledWay:=rAngle, 
	wFS_State:= wFS_State, 
	wCSState:= wGS_State_1,
	wCSState_2:= wGS_State_2,
	xContinue:= xContinue,
	wWaitTillDone:= wGS_WaitTillDone_1, 
	xStartProc:= xGS_StartProc_1, 
	xStartForce:= xFS_Start,
	EndPos:= wGC_EndPos_1, 
	xStartCurve:= xStartAllCurves,
	xStartCurve_2:= xStartAllCurves,  
	xReleaseForce:= xFS_Release, 
	wState=> wST_State_1, 
	rKoef=> , 
	wHalfPos=> );
	
	
CalcDistance(
	wState:= wFS_State, 
	rPos_1:= rTablePos_1, 
	rPos_2:= rTablePos_2, 
	rCyclePos_1:= rAngle, 
	rDistance_1=> rDistance_1, 
	rDistance_2=> rDistance_2, 
	rCycleWay_1=> rFS_CycledWay);
rDistance_1:=fnoneDigit(rDistance_1);
rDistance_2:=fnoneDigit(rDistance_2);	
	
//xST_Ready_1:= wProcType <> 0;
//wST_HalfPos_1:= StiffnessTest.wHalfPos;

END_PROGRAM

// Application/Program/Process/StiffnessTest/fbStiffnessTest
FUNCTION_BLOCK fbStiffnessTest
VAR_INPUT
	xReady			: BOOL;
	rGetForce		: REAL;
	rSetForce		: REAL;
	wGetPos			: DWORD;
	wFS_State		: ForceStepStates;
	wCSState		: CurveStates;
	wCSState_2		: CurveStates;
	wWaitTillDone	: WORD;
	wTyreSizeFirst	: WORD;
	wTyreSizeAfter	: WORD;
	wBufferState_1	: WORD;
	wBufferState_2	: WORD;
	wProcType		: WORD;
	rFS_CycledWay	: REAL;
END_VAR
VAR_IN_OUT
	xStartProc		: BOOL;
	xStartForce		: BOOL;
	xStartCurve		: BOOL;
	xStartCurve_2	: BOOL;
	xReleaseForce	: BOOL;
	EndPos			: WORD;
	xContinue		: BOOL;
END_VAR
VAR_OUTPUT
	wState			: StiffnessTestStates;
	rKoef			: REAL;
	wHalfPos		: DWORD;
	
END_VAR
VAR
	rtStart			: R_TRIG;
	ftStart			: F_TRIG;
	rtGetHalf		: R_TRIG;
	tnWaitTillDone	: TON;	
	HalfPos			: DWORD;
	StartPos		: DWORD;
	tnWait			: TON;
END_VAR

rtStart(CLK:= xStartProc);
ftStart(CLK:= xStartProc);

IF ftStart.Q AND (NOT(wState = ST_Proc_Done)) THEN
	xStartForce		:= FALSE;
	xStartCurve		:= FALSE;
	xStartCurve_2 	:= FALSE;
	xReleaseForce	:= FALSE;
	xContinue		:= FALSE;
	tnWaitTillDone(IN:= FALSE); 
	wState			:= ST_Proc_Stopping;
END_IF


CASE wState OF
	

		ST_Proc_Stop, ST_Proc_Done:
		
				IF xStartProc THEN
					IF wProcType = 4 THEN
						xStartCurve 	:= TRUE;
						xStartCurve_2 	:= TRUE;
						EndPos			:= wTyreSizeFirst;
						wState			:= ST_Proc_GettingFirstCurve;
					ELSIF rFS_CycledWay = 90 THEN
						xStartForce 	:= TRUE;
						wState			:=ST_Proc_GettingForce;
					END_IF
					
					
				END_IF
				
		ST_Proc_GettingFirstCurve:
		
				tnWaitTillDone(IN:= wCSState = CS_Done AND wCSState_2 = CS_Done, PT:= TO_TIME(wWaitTillDone * 1000)); 
				IF tnWaitTillDone.Q THEN
					tnWaitTillDone(IN:= FALSE); 
					xStartCurve 	:= FALSE;
					xStartCurve_2 	:= FALSE;
					//xReleaseForce	:= TRUE;
					//xStartForce 	:= TRUE;
					wState			:=ST_SendingData;
				END_IF
				
				
		ST_SendingData:
		
				IF wCSState_2 = CS_Done AND wBufferState_1 = 0 THEN
					xContinue		:=TRUE;
					wState	:= ST_Proc_Pause;
				END_IF
				
				
		ST_Proc_Pause:
		
				IF (NOT xContinue)THEN
					wState	:= ST_Proc_CalcKoef;
				END_IF
				
				
		ST_Proc_GettingForce:
		
		
				rtGetHalf(CLK:= rGetForce > (rSetForce * 0.5));
				IF rtGetHalf.Q THEN
					wHalfPos := wGetPos - StartPos;
				END_IF
				tnWait(IN:= wFS_State = FS_Done AND rGetForce > (rSetForce * 0.5), PT:=T#5S);
				IF tnWait.Q THEN
					tnWait(IN:=TRUE);
					xReleaseForce	:= TRUE;
					wState	:= ST_Proc_Releasing;
				END_IF
				
				
		ST_Proc_CalcKoef:
		
				tnWaitTillDone(IN:= (*wFS_State = FS_Done AND*) wBufferState_1 = 0 AND wBufferState_2 = 0, PT:= TO_TIME(wWaitTillDone * 1000));
				IF tnWaitTillDone.Q THEN
					tnWaitTillDone(IN:= FALSE); 
					rKoef 			:= (0.5 * rGetForce)/(wGetPos - wHalfPos);
					xStartCurve 	:= TRUE;
					xStartCurve_2 	:= TRUE;
					EndPos			:= wTyreSizeAfter;
					wState		:= ST_Proc_GettingCurve;
				END_IF
				
				
		ST_Proc_GettingCurve:
		
		
				tnWaitTillDone(IN:= wCSState = CS_Done AND wCSState_2 = CS_Done AND wBufferState_1 = 0 AND wBufferState_2 = 0, PT:= TO_TIME(wWaitTillDone * 1000)); 
				IF tnWaitTillDone.Q THEN
					tnWaitTillDone(IN:= FALSE); 
					xStartCurve 	:= FALSE;
					xStartCurve_2 	:= FALSE;
					//xReleaseForce	:= TRUE;
					xStartProc:= FALSE;
					wState			:=ST_Proc_Done;
				END_IF
				

		ST_Proc_Releasing:
				

				IF 	wFS_State = FS_Stop (*AND wBufferState_1 = 0 AND wBufferState_2 = 0 *)THEN
					xStartProc 	:= FALSE;
					wState		:=ST_Proc_Done;
				END_IF
				
		ST_Proc_Stopping:
		
				IF (wFS_State = FS_Stop OR wFS_State = FS_Done) AND (wCSState = CS_Stop OR wCSState = CS_Done) THEN
					wState		:=ST_Proc_Stop;
				END_IF

END_CASE

END_FUNCTION_BLOCK

// Application/Program/Process/StiffnessTest/fbCalcDistance
FUNCTION_BLOCK fbCalcDistance
VAR_INPUT
	wState			: StiffnessTestStates;
	rPos_1			: REAL;
	rPos_2			: REAL;
	rCyclePos_1		: REAL;
END_VAR
VAR_OUTPUT
	rDistance_1			: REAL;
	rDistance_2			: REAL;
	rCycleWay_1			: REAL;
END_VAR
VAR
	rtStart				: R_TRIG;
	rtStop				: R_TRIG;
	rStartPos_1			: REAL;
	rStartPos_2			: REAL;
	rStartCyclePos_1	: REAL;
END_VAR

rtStart(CLK:=wState = FS_FirstRun);
rtStop(CLK:=wState = FS_Done);

IF rtStart.Q THEN
	rStartPos_1			:= rPos_1;
	rStartPos_2			:= rPos_2;
	rStartCyclePos_1	:= rCyclePos_1;
END_IF

//IF rtStop.Q THEN
	IF rPos_1 > rStartPos_1 THEN
		rDistance_1		:= rPos_1 - rStartPos_1;
	ELSE
		rDistance_1		:= rStartPos_1 - rPos_1;
	END_IF
	
	IF rPos_2 > rStartPos_2 THEN
		rDistance_2		:= rPos_2 - rStartPos_2;
	ELSE
		rDistance_2		:= rStartPos_2 - rPos_2;
	END_IF
	
	IF rCyclePos_1 < 300 AND rStartCyclePos_1 < 300 THEN
		IF rCyclePos_1 > rStartCyclePos_1 THEN
			rCycleWay_1	:= rCyclePos_1 - rStartCyclePos_1;
		ELSE
			rCycleWay_1	:= rStartCyclePos_1 - rCyclePos_1;
		END_IF
	ELSIF rCyclePos_1 < 300 THEN
		rCycleWay_1	:= 360 - rStartCyclePos_1 + rCyclePos_1;
	ELSIF rStartCyclePos_1 < 300 THEN
		rCycleWay_1	:= 360 - rCyclePos_1 + rStartCyclePos_1;
	ELSIF rCyclePos_1 > 300 AND rStartCyclePos_1 > 300 THEN
		IF rCyclePos_1 > rStartCyclePos_1 THEN
			rCycleWay_1	:= rCyclePos_1 - rStartCyclePos_1;
		ELSE
			rCycleWay_1	:= rStartCyclePos_1 - rCyclePos_1;
		END_IF
	END_IF
	 
//END_IF

END_FUNCTION_BLOCK

// Application/Program/Process/StiffnessTest/prStiffnessTest_2
PROGRAM prStiffnessTest_2
VAR
	StiffnessTest: fbStiffnessTest;	
END_VAR

StiffnessTest(
	xReady:= xST_Ready_2, 
	rGetForce:= rST_GetForce_2, 
	rSetForce:= rST_SetForce_2, 
	wGetPos:= wFS_ActualPos, 
	wFS_State:= wFS_State, 
	wCSState:= wGS_State_2, 
	wWaitTillDone:= wGS_WaitTillDone_2, 
	xStartProc:= xGS_StartProc_2, 
	xStartForce:= xFS_Start, 
	xStartCurve:= xGC_Start_2, 
	xReleaseForce:= xFS_Release, 
	wState=> wST_State_2, 
	rKoef=> rST_Koef_2, 
	wHalfPos=> wST_HalfPos_2);
	
xST_Ready_2:= wProcType <> 0;
wST_HalfPos_2:= StiffnessTest.wHalfPos;

END_PROGRAM

// Application/Simulation/prSimulation
PROGRAM prSimulation
VAR
	TRAFO:LIN_TRAFO;
	TRAFO_1:LIN_TRAFO;
	Ud : REAL;
	Uv:	REAL;
	ForceStepSim: fbForceStepSim;
	StepperSim_1: fbStepperSim;
	StepperSim_2: fbStepperSim;
END_VAR

 
(*
TRAFO(
	IN:= TO_REAL(Force_Us), 
	IN_MIN:= 0, 
	IN_MAX:= 30000, 
	OUT_MIN:= 0, 
	OUT_MAX:= 15, 
	OUT=> Ud, 
	ERROR=> );
	
	TRAFO_1(
	IN:= TO_REAL(Force_Ref), 
	IN_MIN:= 0, 
	IN_MAX:= 20000, 
	OUT_MIN:= 0, 
	OUT_MAX:= 10, 
	OUT=> Uv, 
	ERROR=> );
rFS_GetForce_check := wFS_ActualPos;
rFS_CycledWay := wFS_ActualPos / 2;

rFS_GetForce:= ((Ud/2)/(Uv))*20000;*)

ForceStepSim(
	xStart:= xFS_Start, 
	xRelease:= xFS_Release, 
	wState=> wFS_State, 
	rActualPosition=> rFS_CycledWay, 
	rActualForce=> rFS_GetForce);
	
StepperSim_1(
	rStartPoint:= 100, 
	rAugment:= -1, 
	xMoveToPos:= xLS_MoveToPos_1, 
	diGetCurve=> rLaserDistance_1, 
	wStepperState=> wLS_StepperState_1);
	
StepperSim_2(
	rStartPoint:= 120, 
	rAugment:= 1, 
	xMoveToPos:= xLS_MoveToPos_2, 
	diGetCurve=> rLaserDistance_2, 
	wStepperState=> wLS_StepperState_2);

END_PROGRAM

// Application/Simulation/fbForceStepSim
FUNCTION_BLOCK fbForceStepSim
VAR_INPUT
	
END_VAR
VAR_IN_OUT
	xStart:				BOOL;
	xRelease:			BOOL;
END_VAR
VAR_OUTPUT
	wState		: ForceStepStates;
	rActualPosition: 	REAL;
	rActualForce:	REAL;
END_VAR
VAR
	tnWait:	TON;
	rtStart:			R_TRIG;
	ftStart:			F_TRIG;
	ftRelease:			F_TRIG;
	rtRelease:			R_TRIG;
END_VAR

rtStart(CLK:=xStart);
ftStart(CLK:=xStart);
rtRelease(CLK:=xRelease);
ftRelease(CLK:=xRelease);

IF (ftStart.Q OR ftRelease.Q)AND (NOT (wState = FS_Done)) THEN	
	xRelease		:= FALSE;	
	wState:=FS_Stop;
END_IF

IF rtRelease.Q THEN
	wState			:=FS_Stop;
END_IF

CASE wState OF
	
	FS_Stop, FS_Done:
	
				IF rtStart.Q THEN										
					wState			:= FS_FirstRun;										
				END_IF
				
	FS_FirstRun:
		
				tnWait(IN:=TRUE, PT:=T#15S);
				rActualPosition:=TO_REAL(tnWait.ET);
				rActualForce:=rActualPosition * 20;
				IF tnWait.Q THEN
					tnWait(IN:=FALSE);
					wState	:= FS_Done;
				END_IF
				

END_CASE

END_FUNCTION_BLOCK

// Application/Simulation/fbStepperSim
FUNCTION_BLOCK fbStepperSim
VAR_INPUT
	rStartPoint:	REAL:=10;
	rAugment: 		REAL:= -2;
END_VAR
VAR_IN_OUT
	xMoveToPos:			BOOL;
END_VAR
VAR_OUTPUT
	diGetCurve:			REAL;
	wStepperState:		StepperStates;
END_VAR
VAR
	rtMoveToPos:		R_TRIG;
	tnWait:				TON;
END_VAR

rtMoveToPos(CLK:=xMoveToPos);

CASE wStepperState OF
	
	SM_Idle, SM_OnPos:
			
								
				IF rtMoveToPos.Q THEN
					diGetCurve:= rStartPoint;
					wStepperState	:= SM_MovingToPos;					
				END_IF
				
	SM_MovingToPos:
			
				
				xMoveToPos		:=FALSE;
				tnWait(IN:= TRUE, PT:=T#2S);
				
				IF tnWait.Q THEN
					tnWait(IN:= FALSE);
					diGetCurve:= rStartPoint + rAugment;
					wStepperState	:= SM_OnPos;
				END_IF
				
				
END_CASE

END_FUNCTION_BLOCK

// Application/Program/Process/GetCurve/prGetCurve_2
PROGRAM prGetCurve_2
VAR
	GetCurve	: fbGetCurve;
	FillBuffer_	: FillBuffer;	
	xStartFilling: BOOL;
	xStopFilling: BOOL;
	xWrite: BOOL;
	xStartSending_2: BOOL;
	ConturBuffer_:	ConturBuffer;
	rtStopFilling:	R_TRIG;
	ReadBuffOPC: fbReadBuffOPC;
	xStopSending: BOOL;
	rtStopSending_:	R_TRIG;
END_VAR

GetCurve(
	diDistance:= wGC_Distance_2, 
	rGetPos:= rLS_RealPos_2,
	wStepperState:= wLS_StepperState_2, 
	xInitilized:= xLS_Initilized_2, 
	wInitialPos:= 50,
	xReadOPC:=	xWrite,//wGC_InitialPos_2, 
	wEndPos:= wGC_EndPos_2,
	xCurveStarted:=xCurveStarted_2,  
	xStart:= xGC_Start_2, 
	xMovePos:= xLS_MoveToPos_2, 
	xStopStep:= xLS_Stop_2, 
	wSetPos:= wLS_SetPos_2, 
	wState=> wGS_State_2);
	
	
IF xCurveStarted_2 THEN
	xStartFilling:=	TRUE;
END_IF

rtStopFilling(CLK:=wGS_State_2 = CS_Done);
IF rtStopFilling.Q THEN
	xStopFilling:= TRUE;
END_IF

rtStopSending_(CLK:=wGS_State_2 = CS_Stop);
IF rtStopSending_.Q THEN
	xStopSending:=TRUE;
END_IF
	
FillBuffer_(
	rStepPos:= rLS_RealPos_2, 
	rLaserData:= rLaserDistance_2, 
	xStart:= xStartFilling, 
	xStop:= xStopFilling, 
	xWrite:= xWrite,
	xStartSending:= xStartSending_2,  
	ConturBuffer=> ConturBuffer_);

ReadBuffOPC(
	ConturBuffer:= ConturBuffer_, 
	wIndexOfReadynnes:= 5, 
	xStart:= xStartSending_2, 
	xSend:= xReadOPC_2,
	xStop:= xStopSending, 
	rStepPos=> rStepPos_2,
	rLaserData=> rLaserData_2, 
	wState=> );

END_PROGRAM
